// TIA Portal project "Soru6" (V15)

(* hardware
DEVICE "S7-1200 station_1"  S7-1200 Station
   slot 0: "Rack_0"  S7-1200 Rack  Rack  V1.0
   slot 1: "PLC_1"  CPU 1214C DC/DC/DC  6ES7 214-1AG40-0XB0  V4.2
*)

// ===== PLC "PLC_1"  CPU 1214C DC/DC/DC =====

VAR_GLOBAL   // PLC tag table "Default tag table"
   "Dudur" AT %I0.0 : Bool;
   "Basla" AT %I0.1 : Bool;
   "optikSenosr" AT %I0.2 : Bool;
   "konvoyor_1" AT %Q0.0 : Bool;
   "konvoyor_2" AT %Q0.1 : Bool;
   "Deger" AT %MD0 : DWord;
   "Kalan_icin" AT %MD4 : DWord;
END_VAR

// folder: System blocks/Program resources

DATA_BLOCK "zmn1"   // DB1
{ S7_Optimized_Access := 'TRUE' }
AUTHOR : Simatic
FAMILY : IEC
NAME : IEC_TMR
VERSION : 1.0
// stored: InstanceOfName IEC_TIMER
"IEC_TIMER"
BEGIN
END_DATA_BLOCK

DATA_BLOCK "zmn2"   // DB2
{ S7_Optimized_Access := 'TRUE' }
AUTHOR : Simatic
FAMILY : IEC
NAME : IEC_TMR
VERSION : 1.0
// stored: InstanceOfName IEC_TIMER
"IEC_TIMER"
BEGIN
END_DATA_BLOCK

DATA_BLOCK "sayac"   // DB3
{ S7_Optimized_Access := 'TRUE' }
AUTHOR : Simatic
FAMILY : IEC
NAME : UCNTR
VERSION : 1.2
// stored: InstanceOfName IEC_UCOUNTER
"IEC_UCOUNTER"
BEGIN
END_DATA_BLOCK

DATA_BLOCK "ardisik"   // DB4
{ S7_Optimized_Access := 'TRUE' }
AUTHOR : Simatic
FAMILY : IEC
NAME : UCNTR
VERSION : 1.2
// stored: InstanceOfName IEC_UCOUNTER
"IEC_UCOUNTER"
BEGIN
END_DATA_BLOCK

// folder: (top level)

ORGANIZATION_BLOCK "Main"   // OB1, LAD, ProgramCycle
TITLE = "Main Program Sweep (Cycle)"
{ S7_Optimized_Access := 'TRUE' }
VERSION : 0.1
   VAR_INPUT
      Initial_Call : Bool;   // Initial call of this OB
      Remanence : Bool;   // =True, if remanent data are available
   END_VAR
BEGIN

REGION Network 1: Zman döngüsü
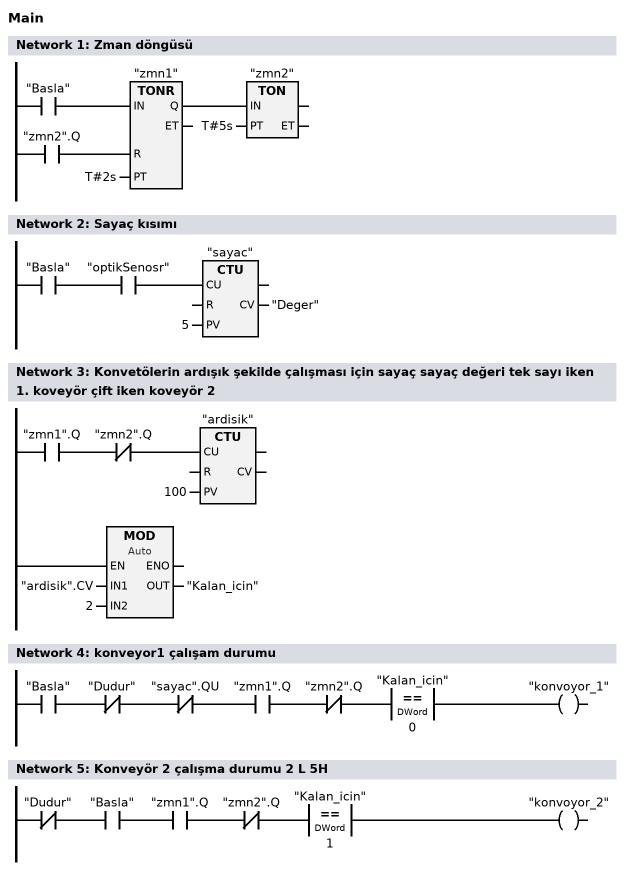
   "zmn1".TONR(IN := "Basla", R := "zmn2".Q, PT := T#2s);
   "zmn2".TON(IN := "zmn1".Q, PT := T#5s);
END_REGION

REGION Network 2: Sayaç kısımı
   "sayac".CTU(CU := "Basla" AND "optikSenosr", PV := 5, CV => "Deger");
END_REGION

REGION Network 3: Konvetölerin ardışık şekilde çalışması için sayaç sayaç değeri tek sayı iken 1. koveyör çift iken koveyör 2
   "ardisik".CTU(CU := "zmn1".Q AND NOT "zmn2".Q, PV := 100);
   "Kalan_icin" := "ardisik".CV MOD 2;
END_REGION

REGION Network 4: konveyor1 çalışam durumu
   RUNG wire#powerrail
      Contact( "Basla" )
      I_Contact( "Dudur" )
      I_Contact( "sayac".QU )
      Contact( "zmn1".Q )
      I_Contact( "zmn2".Q )
      { S7_Templates := "SrcType := DWord" } EQ_Contact(in1 := "Kalan_icin", in2 := 0)
      Coil( "konvoyor_1" )
   END_RUNG
   // the same network as SCL:
   "konvoyor_1" := "Basla" AND NOT "Dudur" AND NOT "sayac".QU AND "zmn1".Q AND NOT "zmn2".Q AND ("Kalan_icin" = 0);
END_REGION

REGION Network 5: Konveyör 2 çalışma durumu 2 L 5H
   RUNG wire#powerrail
      I_Contact( "Dudur" )
      Contact( "Basla" )
      Contact( "zmn1".Q )
      I_Contact( "zmn2".Q )
      { S7_Templates := "SrcType := DWord" } EQ_Contact(in1 := "Kalan_icin", in2 := 1)
      Coil( "konvoyor_2" )
   END_RUNG
   // the same network as SCL:
   "konvoyor_2" := NOT "Dudur" AND "Basla" AND "zmn1".Q AND NOT "zmn2".Q AND ("Kalan_icin" = 1);
END_REGION
END_ORGANIZATION_BLOCK